// TwinCAT 3 PLC project PLC
// ProgramVersion: 3.1.4023.0
// libraries:
//   Tc2_Standard, * (Beckhoff Automation GmbH)
//   Tc2_System, * (Beckhoff Automation GmbH)
//   Tc3_Module, * (Beckhoff Automation GmbH)
// project tree:
//   / PlcTask.TcTTO
//   POUs/ FbCalculator.TcPOU, MAIN.TcPOU
// real-time tasks:
//   TASK PlcTask: cycle T#10ms, priority 20, ADS port 350

CONFIGURATION PLC
    RESOURCE PLC ON TwinCAT3
        TASK PlcTask(INTERVAL := T#10ms, PRIORITY := 20);
        PROGRAM MAIN WITH PlcTask : MAIN;
    END_RESOURCE
END_CONFIGURATION

// ---- POUs/MAIN.TcPOU
PROGRAM MAIN
VAR
    _fbCalculator : FbCalculator;
END_VAR

END_PROGRAM

// ---- POUs/FbCalculator.TcPOU
FUNCTION_BLOCK FbCalculator
VAR_INPUT
END_VAR
VAR_OUTPUT
END_VAR
VAR
END_VAR

{attribute 'TcRpcEnable'}
METHOD PUBLIC Sum : LREAL
VAR_INPUT
    Input1 : LREAL;
    Input2 : LREAL;
END_VAR
Sum := Input1 + Input2;
END_METHOD

END_FUNCTION_BLOCK
